FUNCTION_BLOCK LD_XOR (* Ladder Diagram XOR function *)
  (* Standard: 61499-2 *)
  (* Version 0.3, 2006-09-06, JHC, Holobloc Inc, Made a SimpleFB *)
  (* Version 0.2, 2003-12-04, JHC, Rockwell Automation, Renamed for better indexing. *)
  (* Version 0.1, 2002-11-05, JHC, Rockwell Automation, Corrected missing ST element in Algorithm REQ. *)
  (* Version 0.0, 2000-05-30, JHC, Rockwell Automation *)
  (* Compiler header: package fb.rt.student; *)
  (* Compiler classdef: SimpleFB *)
  (* Compiler Java Sun JDK 1.5.0 *)
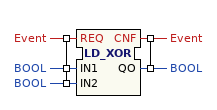
  EVENT_INPUT
    REQ WITH IN1, IN2; (* Normal Execution Request *)
  END_EVENT
  EVENT_OUTPUT
    CNF WITH QO; (* Execution Confirmation *)
  END_EVENT
  VAR_INPUT
    IN1 : BOOL;
    IN2 : BOOL;
  END_VAR
  VAR_OUTPUT
    QO : BOOL; (* IN1 XOR IN2 *)
  END_VAR
  ALGORITHM REQ IN LD: (* Normally executed algorithm *)
    QO := IN1 IN2 ! & IN1 ! IN2 & |;
  END_ALGORITHM
END_FUNCTION_BLOCK
